{attribute 'pack_mode' := '1'} 
FUNCTION_BLOCK FB_Packed
VAR_INPUT
	bMember	: T_Bool := TRUE;
	nMember : T_Dint := -57;
	sMember : STRING := 'Testing Error.';
END_VAR

END_FUNCTION_BLOCK

(* stored: Version 1.1.0.1
   POU FB_Packed: Id {5bb1f1cf-d4c9-40dc-915a-25d6b054702a}, SpecialFunc None *)
